# EPICS substitutions: iocBoot/ioc-tst-gige-01/ioc-tst-gige-01.substitutions
#
# unixCam IOC archive substitutions file
#

# Generate generic portion of unixCam archive request
file archive_gige.archive
{
    {
        IOC     =   TST:R40:IOC:18:GIGE:01,
    }
}
